(* PLC project PLC, Beckhoff Automation GmbH TwinCAT PLC Control 3.5.13.21 *)
(* stored: creationDateTime 2024-02-17T22:40:51.1336007, modificationDateTime 2024-02-17T22:40:51.1366008 *)

TYPE CylConfig :
STRUCT
	operateDelayTime: TIME;
	sensorDelayTime: TIME;
	cylinderErrorTime: TIME;
END_STRUCT
END_TYPE

TYPE CylInput :
STRUCT
	posFw AT %I*: BOOL;
	posRv AT %I*: BOOL;
END_STRUCT
END_TYPE

TYPE CylOutput :
STRUCT
	opeFw AT %Q*: BOOL;
	opeRv AT %Q*: BOOL;
END_STRUCT
END_TYPE

TYPE CylResource :
STRUCT
	input: CylInput;
	output: CylOutput;
	config: CylConfig;
	status: CylStatus;
END_STRUCT
END_TYPE

TYPE CylStatus :
STRUCT
	name: STRING(G.nameStringLength);
	opeFw: BOOL;
	opeRv: BOOL;
	posFw: BOOL;
	posRv: BOOL;
	ready: BOOL;
	busy: BOOL;
	done: BOOL;
	error: BOOL;
	errorCode: LINT;
	opePastTime: TIME;
END_STRUCT
END_TYPE

TYPE PBInput :
STRUCT
	pushed AT %I*: BOOL;
END_STRUCT
END_TYPE

TYPE PBStatus :
STRUCT
	name: STRING(G.nameStringLength);
	pushed: BOOL;
END_STRUCT
END_TYPE

TYPE PBResource :
STRUCT
	input: PBInput;
	config: PBConfig;
	status: PBStatus;
END_STRUCT
END_TYPE

TYPE PBConfig :
STRUCT
	pushDelayTime: TIME;
END_STRUCT
END_TYPE

TYPE LPConfig :
STRUCT
	invert: BOOL;
END_STRUCT
END_TYPE

TYPE LPStatus :
STRUCT
	name: STRING(G.nameStringLength);
	on: BOOL;
END_STRUCT
END_TYPE

TYPE LPOutput :
STRUCT
	on AT %Q*: BOOL;
END_STRUCT
END_TYPE

TYPE LPResource :
STRUCT
	output: LPOutput;
	config: LPConfig;
	status: LPStatus;
END_STRUCT
END_TYPE

FUNCTION_BLOCK Cyl
VAR_INPUT
	index: LINT;
	name: STRING(G.nameStringLength);
	opeFw: BOOL;
	opeRv: BOOL;
END_VAR
VAR_OUTPUT
	posFw: BOOL;
	posRv: BOOL;
	ready: BOOL;
	busy: BOOL;
	done: BOOL;
	error: BOOL;
END_VAR
VAR_IN_OUT
	resources: ARRAY[0..G.numAxis] OF CylResource;
END_VAR
VAR
	input: CylInput;
	output: CylOutput;
	config: CylConfig;
	status: CylStatus;
	rsErrorON: BOOL;
	rsErrorOFF: BOOL;
	cylErrorFw: BOOL;
	cylErrorRv: BOOL;
	TON_0: TON;
	TON_1: TON;
	TON_2: TON;
	TON_3: TON;
	TON_4: TON;
	TON_5: TON;
END_VAR

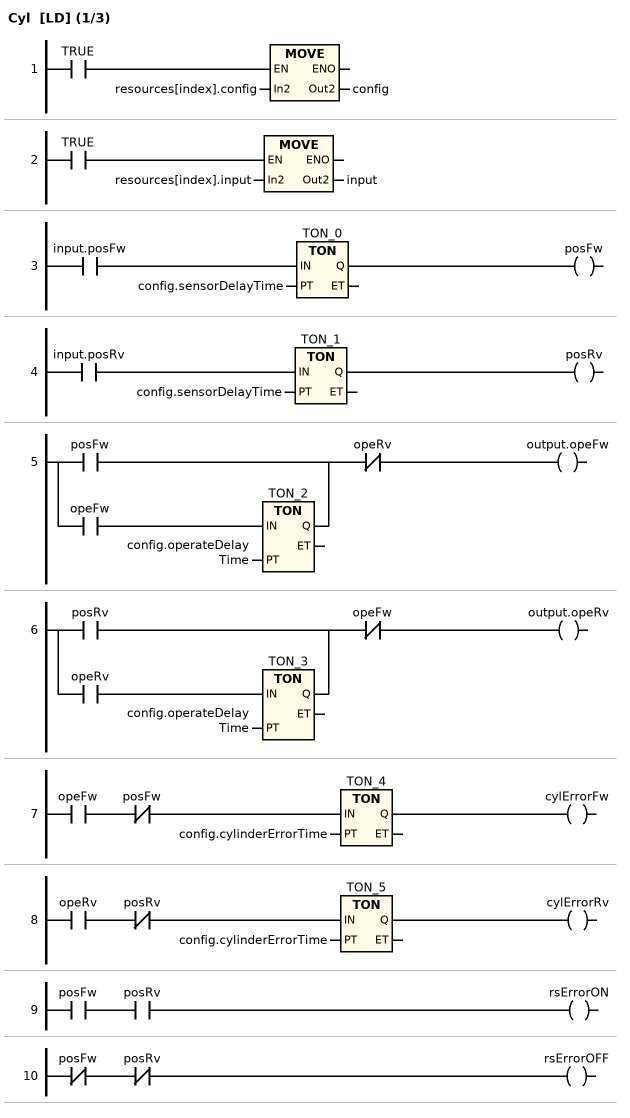
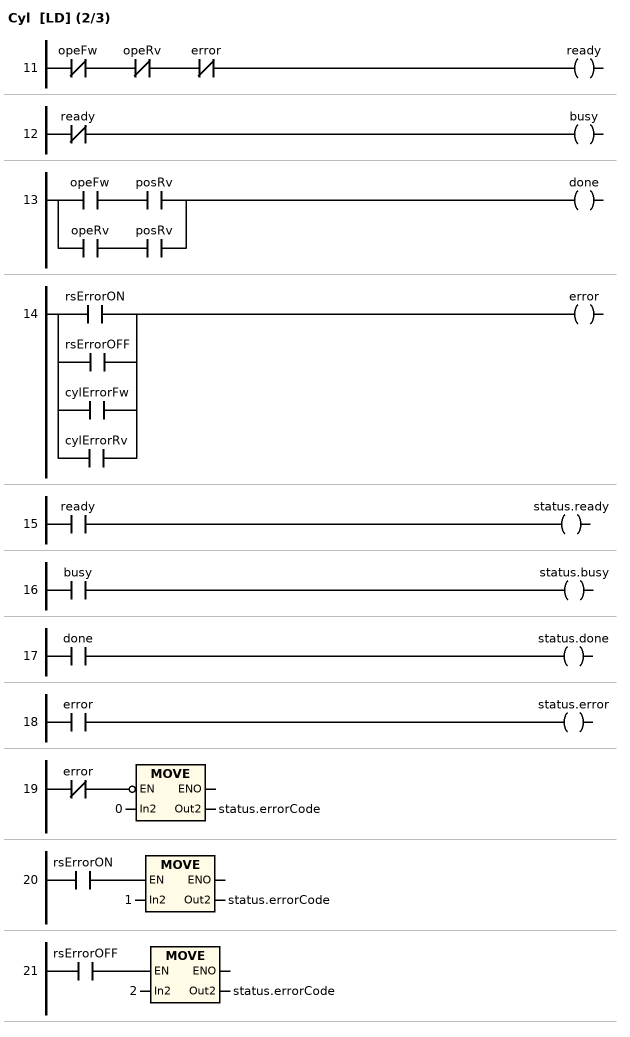
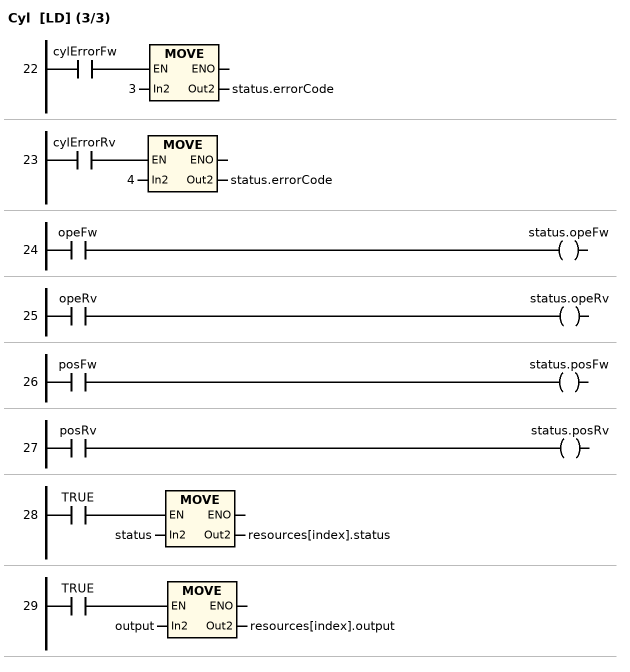
(* LD diagram, written out as Structured Text *)

IF TRUE THEN config := resources[index].config; END_IF;

IF TRUE THEN input := resources[index].input; END_IF;

TON_0(IN := input.posFw, PT := config.sensorDelayTime);
posFw := TON_0.Q;

TON_1(IN := input.posRv, PT := config.sensorDelayTime);
posRv := TON_1.Q;

TON_2(IN := opeFw, PT := config.operateDelayTime);
output.opeFw := (TON_2.Q OR posFw) AND NOT opeRv;

TON_3(IN := opeRv, PT := config.operateDelayTime);
output.opeRv := (TON_3.Q OR posRv) AND NOT opeFw;

TON_4(IN := opeFw AND NOT posFw, PT := config.cylinderErrorTime);
cylErrorFw := TON_4.Q;

TON_5(IN := opeRv AND NOT posRv, PT := config.cylinderErrorTime);
cylErrorRv := TON_5.Q;

rsErrorON := posFw AND posRv;

rsErrorOFF := NOT posFw AND NOT posRv;

ready := NOT opeFw AND NOT opeRv AND NOT error;

busy := NOT ready;

done := opeFw AND posRv OR opeRv AND posRv;

error := rsErrorON OR rsErrorOFF OR cylErrorFw OR cylErrorRv;

status.ready := ready;

status.busy := busy;

status.done := done;

status.error := error;

IF NOT (NOT error) THEN status.errorCode := 0; END_IF;

IF rsErrorON THEN status.errorCode := 1; END_IF;

IF rsErrorOFF THEN status.errorCode := 2; END_IF;

IF cylErrorFw THEN status.errorCode := 3; END_IF;

IF cylErrorRv THEN status.errorCode := 4; END_IF;

status.opeFw := opeFw;

status.opeRv := opeRv;

status.posFw := posFw;

status.posRv := posRv;

IF TRUE THEN resources[index].status := status; END_IF;

IF TRUE THEN resources[index].output := output; END_IF;
(* --- network --- *)
END_FUNCTION_BLOCK

PROGRAM MAIN
VAR
	// resources
	cylinders: ARRAY[0..G.numAxis] OF CylResource;
	PBs: ARRAY[0..G.numAxis] OF PBResource;
	LPs: ARRAY[0..G.numAxis] OF LPResource;
	
	// system
	firstScan: BOOL := TRUE;
	
	// 動作設定
	permConfigCyl: ARRAY[0..G.numAxis] OF CylConfig;
	permConfigPB: ARRAY[0..G.numAxis] OF PBConfig;
	permConfigLP: ARRAY[0..G.numAxis] OF LPConfig;
	i: LINT;
	unmatchConfig: BOOL := FALSE;
END_VAR

                  Unit();


// 動作設定不一致を調べる
unmatchConfig := FALSE;
FOR i := 0 TO G.numAxis DO
	IF permConfigCyl[i].cylinderErrorTime <> cylinders[i].config.cylinderErrorTime THEN
		unmatchConfig := TRUE;
	END_IF
	IF permConfigCyl[i].operateDelayTime <> cylinders[i].config.operateDelayTime THEN
		unmatchConfig := TRUE;
	END_IF
	IF permConfigCyl[i].sensorDelayTime <> cylinders[i].config.sensorDelayTime THEN
		unmatchConfig := TRUE;
	END_IF
	IF permConfigPB[i].pushDelayTime <> PBs[i].config.pushDelayTime THEN
		unmatchConfig := TRUE;
	END_IF
	IF permConfigLP[i].invert <> LPs[i].config.invert THEN
		unmatchConfig := TRUE;
	END_IF
END_FOR


// 起動後初回に動作設定を元に戻す
IF firstScan THEN
	FOR i := 0 TO G.numAxis DO
		cylinders[i].config := permConfigCyl[i];
		PBs[i].config := permConfigPB[i];
		LPs[i].config := permConfigLP[i];
	END_FOR
END_IF


firstScan := FALSE;
                
END_PROGRAM

PROGRAM Unit
VAR
	stopperToUp: BOOL;
	stopperToDown: BOOL;	

	stopper: Cyl;
	fwButton: PB;
	rvButton: PB;
	
	unmatchConfigLamp: LP;
END_VAR

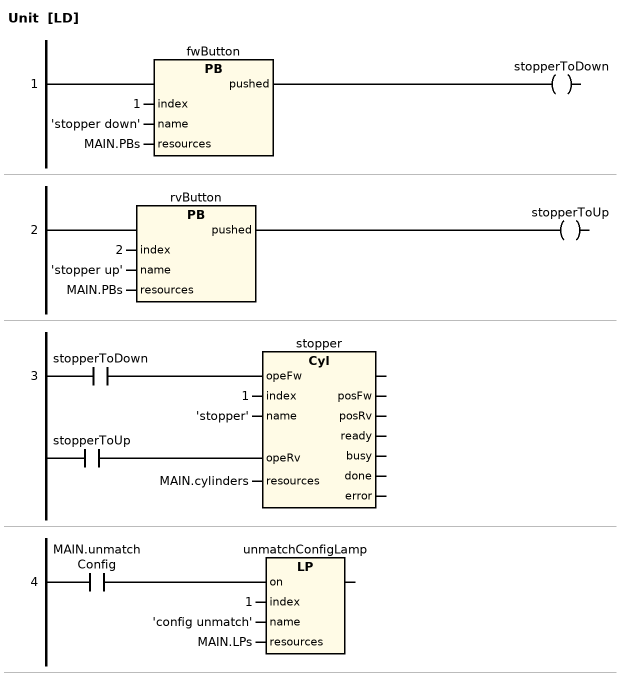
(* LD diagram, written out as Structured Text *)

fwButton(index := 1, name := 'stopper down', resources := MAIN.PBs);
stopperToDown := fwButton.pushed;

rvButton(index := 2, name := 'stopper up', resources := MAIN.PBs);
stopperToUp := rvButton.pushed;

stopper(index := 1, name := 'stopper', opeFw := stopperToDown, opeRv := stopperToUp, resources := MAIN.cylinders);

unmatchConfigLamp(index := 1, name := 'config unmatch', on := MAIN.unmatchConfig, resources := MAIN.LPs);
END_PROGRAM

FUNCTION_BLOCK PB
VAR_INPUT
	index: LINT;
	name: STRING(G.nameStringLength);
END_VAR
VAR_OUTPUT
	pushed: BOOL;
END_VAR
VAR_IN_OUT
	resources: ARRAY[0..G.numAxis] OF PBResource;
END_VAR
VAR
	input: PBInput;
	config: PBConfig;
	status: PBStatus;
	TON_0: TON;
END_VAR

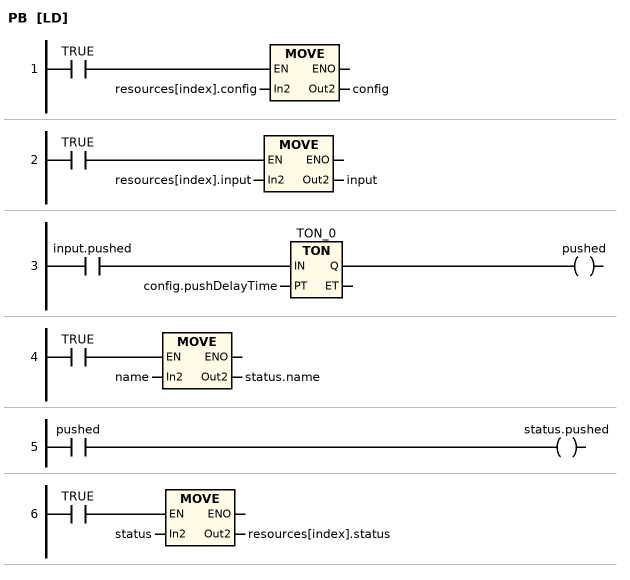
(* LD diagram, written out as Structured Text *)

IF TRUE THEN config := resources[index].config; END_IF;

IF TRUE THEN input := resources[index].input; END_IF;


TON_0(IN := input.pushed, PT := config.pushDelayTime);
pushed := TON_0.Q;

IF TRUE THEN status.name := name; END_IF;

status.pushed := pushed;

IF TRUE THEN resources[index].status := status; END_IF;
END_FUNCTION_BLOCK

FUNCTION_BLOCK LP
VAR_INPUT
	index: LINT;
	name: STRING(G.nameStringLength);
	on: BOOL;
END_VAR
VAR_OUTPUT
END_VAR
VAR_IN_OUT
	resources: ARRAY[0..G.numAxis] OF LPResource;
END_VAR
VAR
	output: LPOutput;
	config: LPConfig;
	status: LPStatus;
END_VAR

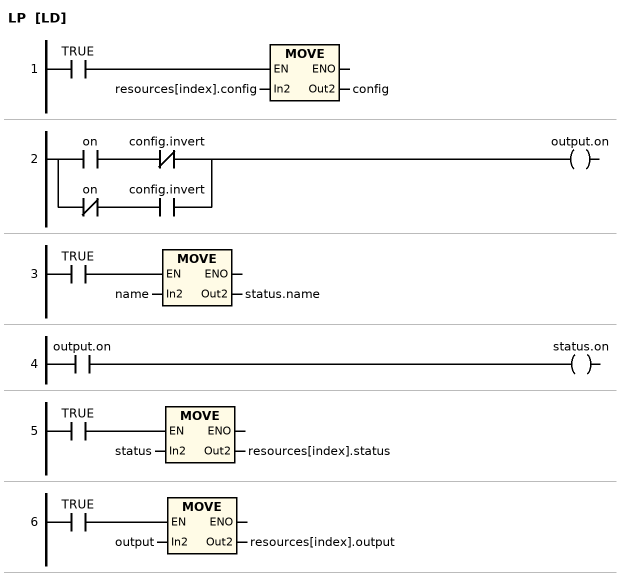
(* LD diagram, written out as Structured Text *)

IF TRUE THEN config := resources[index].config; END_IF;

output.on := on AND NOT config.invert OR NOT on AND config.invert;

IF TRUE THEN status.name := name; END_IF;

status.on := output.on;

IF TRUE THEN resources[index].status := status; END_IF;

IF TRUE THEN resources[index].output := output; END_IF;
(* --- network --- *)
END_FUNCTION_BLOCK

CONFIGURATION Application
  RESOURCE PLC ON PLC
(* global variable list G *)
{attribute 'qualified_only'}
VAR_GLOBAL CONSTANT
	numAxis: LINT := 128;
	nameStringLength: LINT := 64;
END_VAR
VAR_GLOBAL
END_VAR
    TASK PlcTask(INTERVAL := T#0ms, PRIORITY := 20);
    PROGRAM MAIN WITH PlcTask : MAIN;
  END_RESOURCE
END_CONFIGURATION
